// TIA Portal V20 export
FUNCTION "RealBlockName" : Void   // FC17, LAD
BEGIN

REGION Network 1
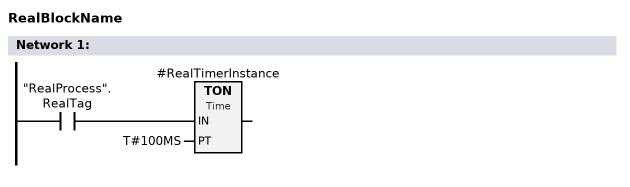
   RUNG wire#powerrail
      Contact( "RealProcess".RealTag )
      { S7_Templates := "time_type := Time" } #RealTimerInstance.TON(pt := T#100MS)
   END_RUNG
   // the same network as SCL:
   #RealTimerInstance.TON(IN := "RealProcess".RealTag, PT := T#100MS);
END_REGION
END_FUNCTION
